{attribute 'linkalways'} 
{attribute 'no_explicit_call' := 'This FB is a CLASS and must be accessed using methods or properties'}
{attribute 'enable_dynamic_creation'}
FUNCTION_BLOCK FINAL MAX_SINT EXTENDS Node
VAR
	in1 : _SINT(0);
	in2 : _SINT(0);
	out : _SINT(0);
END_VAR

METHOD PUBLIC Clone : I_Node
VAR
	pNode : POINTER TO MAX_SINT;
END_VAR
pNode := __NEW(MAX_SINT);
Clone := pNode^;
END_METHOD

METHOD FB_init : BOOL
VAR_INPUT
	bInitRetains : BOOL; // if TRUE, the retain variables are initialized (warm start / cold start)
	bInCopyCode : BOOL;  // if TRUE, the instance afterwards gets moved into the copy code (online change)
END_VAR
AddInput('in1',THIS^.in1);
AddInput('in2',THIS^.in2);
AddOutput('out', THIS^.out);
END_METHOD

METHOD PROTECTED OnExecute
VAR
END_VAR
out.Value := MAX(in1.Value, in2.Value);
END_METHOD

END_FUNCTION_BLOCK

(* stored: Version 1.1.0.1, ProductVersion 3.1.4024.15
   POU MAX_SINT: Id {c3ffb006-eae5-4765-94a5-2fd3035b0723}, SpecialFunc None
   Folder Constructor: Id {4d767815-5d40-4666-8d02-33745b7cee34}
   Method Clone: Id {b5af0143-8182-433c-b58c-474988817f58}
   Method FB_init: Id {0b4367fb-645f-4cfe-a179-f31844f4e388}
   Method OnExecute: Id {96750b85-4d6d-4df7-9c73-bef5c3bef9b0} *)
